# B&R Automation Studio project DeltaTracking
Automation Studio 6.5.1.6; technology packages: mappCockpit 6.3.1, mappMotion 6.6.0, mappView 6.3.0, OpcUaCs 6.0.0

## Configuration Config1

CPU 5APC3100.KBU3-000, AutomationRuntime 6.6.3, Build 11.3.0, Safety 0.0

### Task classes (Cpu.sw)
```
Cyclic#1 (cycle 2000 us, tolerance 0 us):
  APP_Convey <- Conveyor.APP_Conveyor1.prg
  APP_Robot1 <- Robots.APP_Robot1.prg
DataObjects: Arnc0sys, Acp10sys
NcDataObjects: gmcipuc, gmciplog, gmcipfub, gmcipfun, gmciplsm, gmciplbr, gmcipmxd, gmcipvar, gmcipsys, gmcipiec, gmcipesm, gmcipusm, gmcipcsm, gmcipui, gmcipubr, gmcipcbr, gmcipcfg, gmcipus, gmcipmx, Cam
Binaries: McAcpSys, mcdrivelog, udbdef, TCData, mvLoader, arsvcreg, arflatprv, mCoWebSc, McAcpDrv, McAcpSim, McProfGen, McMechSys, arcoal, ashwac, arconfig, asfw, ashwd, iomap, User, Role, sysconf, TraceConfi, Settings, Config_1, Hierarchy, Config, AxisAx_1, Config_2, ComRobot, Config_4, Config_5, Config_3, Config_6, ToolX20, AxesAxX21, GRobot1, GFRobot1, ARobot1, ComRobot1, WorkRobot1, GRobot2, MRobot1, GFRobot2, FeatX21, TrkDevX21, TrkDevConv, AxisAxX25, MecX20, AxesAxX20, WorkX20, FeatX20, DeltaX20, ComFeatX20, DeltaX21, TrkDevX20, vccddbox, vcfile, vccbtn, vcpdvnc, arialbd, vcmgr, vctcal, vcgclass, vcctext, vccnum, vcfntttf, vcdsloc, vccstr, arial, Visu03, vccshape, vcalarm, Visu01, vccdt, vccscale, vcchtml, vcchspot, vccbmp, vccpopup, vcshared, vcxml, vccurl, vcrt, vccslider, Visu02, vcnet, vcclbox, vcbclass, vcdsint, vcpdsw, vccovl, vccline, TCLang, visvc, vccdbox, vcpfar00, vcpfmtcx, vcpfapc, GrpMaster, Users, UsersLogin, TC, Files, DiagWebXs, AlmMaster, AlmHisMain, AlmMain, GrpVMaster, AlmVMaster, CfgPureVir, AxisPS, AxisAxXX1, AxisAxXX2, AxisMaster, MDevXX1, AxVMaster, GrpDevXX1, AlmDevXX1, GrPDevXX4, AlmDevXX4, GrPDevX10, AlmDevX10, AlmDevX20, GrpDevX20, AlmDevX21, GrpDevX21, AlmMBelts, GrpMBelts, AlmDevXX6, GrpDevXX6, AxesVAxX20, vcpfx20, AxisMBelts, MasMBelts, MBeltsPt, AxesVAxX25, AxesAxX10, AxesAxX25, WorkX10, CncXX6, MecX10, AxesVAxX10, DeltaX10, FeatXX6, FeatX10, ToolX10, ToolXX6, MecXX6, MotMaster, MotVMaster, vcctrend, MotDevX10, GrPDevXX3, AlmDevXX3, MotDevXX3, GrPDevXX2, MotDevXX1, AlmDevXX2, MotDevXX2, vcpkat, arnc0cfg, Sdc10map, Arnc0map, Sdc10map1, Sdc10map2, MotDevX20, MotDevX11, MotDevXX9, GrpDevXX9, AlmDevXX9, PML, MotDevXX6, CncDevXX6, MotDevXX7, AlmDevXX7, GrpDevXX7, Robot, AlmDevXX8, GrpDevXX8, MotSim, MotSpindle, MotDevXXA, AlmDevXXA, GrpDevXXA, GrpDevX11, AlmDevX11, OpcUaBasic, User_1, OpcUaMap, AlmHmi, AlmHistHmi, Groups, vccpiech, MotMac, acp10cfg, Acp10map
Libraries: standard, AsBrStr, sys_lib, runtime, AsArSdm, astime, brsystem, FileIO, AsIODiag, DataObj, AsArProf, AsMem, AsIOAcc, AsEPL, ASMcDcs, AsBrMath, visapi, ArTextSys, AsSem, AsIecCon, AsZip, powerlnk, aruser, asusb, ashw, arcert, arssl, aseth, asio, vcresman, IecCheck, areventlog, MpCom, MpUserX, MpFile, MpRecipe, MpAlarmX, MpBase, CoTrace, MpServer, McBase, McAxGroup, McAcpAx, McAxis, McPathGen, McTrkPath, MpAxis, McProgInt, McPureVAx, McDS402Ax, MpRobotics, MpCnc, MpTool
```

### Hardware
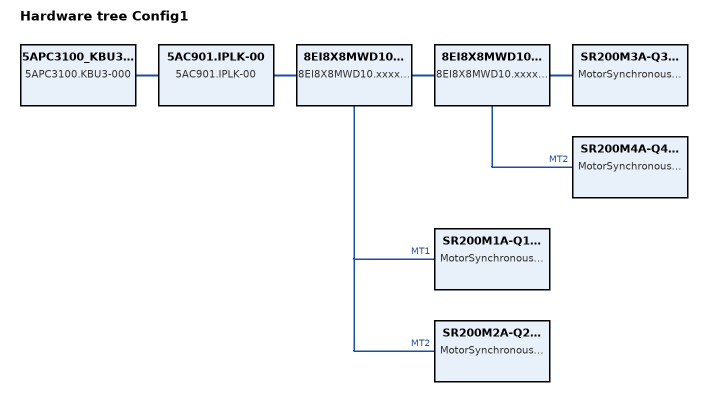
```
5AC901.IPLK-00 : 5AC901.IPLK-00 v2.1.0.0  [SL -> 5APC3100_KBU3_000.SL2]
  Connector IF1:
    DNAConfiguration = manual
    Channel1
    ChannelID1 = McAcpBroadcast
    ChannelType1 = OCTET[96]
5APC3100_KBU3_000 : 5APC3100.KBU3-000 v2.3.1.0
  Connector IF3:
    AssignedOperatingSystem = ARemb
    ActivateDevice = 1
    HostName = apc3100robert
    Mode = Manual
    InternetAddress = 10.43.51.43
    SubnetMask = 255.255.255.0
    Vnc1
    VncKeyMappingFile1 = 
    VncRefreshRate1 = 100
    ActivateSnmp = 2
  Connector IF4:
    AssignedOperatingSystem = ARemb
    ActivateDevice = 1
    HostName = apc3100robert
    Mode = DHCPServer
    InternetAddress = 192.168.20.254
    SubnetMask = 255.255.255.0
    Lease1
    LeaseName1 = Range1
    LeaseStartAddress1 = 192.168.20.100
    LeaseStopAddress1 = 192.168.20.110
    LeaseSubnetMask1 = 255.255.255.0
    Vnc1
    VncTitle1 = VNC
    ActivateSnmp = 2
  Connector IF5:
    AssignedOperatingSystem = ARemb
  Connector IF6:
    AssignedOperatingSystem = ARemb
  Connector IF7:
    AssignedOperatingSystem = ARemb
  Connector IF8:
    AssignedOperatingSystem = ARemb
  ConfigurationID = Template_X20CP1586
  UserPartitionSize = 5
  Simulation = 1
  TimerDeviceType = EPLX2X
  TimerDevice = 5AC901.IPLK-00.IF1
  IdleTaskClass = 4
  TaskClassIdleTime = 4000
  Cyclic1Duration = 2000
  Cyclic1Tolerance = 0
  Cyclic1Stack = 16384
  Cyclic2Duration = 4000
  Cyclic2Tolerance = 0
  Cyclic3Duration = 10000
  Cyclic3Tolerance = 0
  Cyclic4Duration = 20000
  Cyclic4Tolerance = 0
  Cyclic5Duration = 50000
  Cyclic5Tolerance = 0
  Cyclic6Duration = 100000
  Cyclic6Tolerance = 0
  Cyclic7Duration = 200000
  Cyclic7Tolerance = 0
  FileDevice1
  FileDeviceName1 = SceneViewer
  FileDevicePath1 = USER_PATH
  FileDevice2
  FileDeviceName2 = MPLogDir
  FileDevicePath2 = USER_PATH\Log
  FileDevice3
  FileDeviceName3 = DebugData
  FileDevicePath3 = USER_PATH\\Debug
  FileDevice4
  FileDeviceName4 = CNC_PrgDir
  FileDevicePath4 = USER_PATH\CNC_Prg
  EthernetDefaultGateway = 10.43.51.1
  ActivateFtpServer = 1
  FTPProtocol = 2
  FtpUser1
  FtpUsername1 = gmctest
  FtpUserPassword1 = dJg12F/7hd2fGO/QauVo5qNTeUud8LRwkPqca2btE1Q=
  FtpUserSalt1 = iGhlfz5v
  FTPAccessRight1 = 0
  FTPdevice1 = ALL
  ActivateWebServer = 1
  ActivateSdm = 1
8EI8X8MWD10.xxxx-1-Q1-Q2_SRr500_1 : 8EI8X8MWD10.xxxx-1 v2.4.0.0 (NodeNumber=1)  [PLK1 -> 5AC901.IPLK-00.IF1 [Cable Type=PowerlinkCable, Length=10, Version=1.0.0.3]; PLK2 -> 8EI8X8MWD10.xxxx-1-Q3-Q4_SRr500_1.PLK1 [Cable Type=PowerlinkCable, Length=10, Version=1.0.0.3]; MT2 -> SR200M2A-Q2_SRr500_1.MT]
  DriveConfiguration/Encoder/EncoderX41:
    InterfaceType = T_Format
  DriveConfiguration/Encoder/EncoderX42:
    InterfaceType = T_Format
  DriveConfiguration/Channel[1]/RealAxis:
    AxisReference = gAxisQ1_SRr500_1
  DriveConfiguration/Channel[1]/RealAxis/MechanicalElements/Gearbox:
    InputIsReadOnly = 1
    Input = 80
    OutputIsReadOnly = 1
  DriveConfiguration/Channel[1]/RealAxis/MechanicalElements/RotaryToLinearTransformation:
    ReferenceDistanceIsReadOnly = 1
    ReferenceDistance = 360
  DriveConfiguration/Channel[1]/RealAxis/Controller:
    ModeIsReadOnly = 1
    Mode = PositionControllerWithTorqueFeedForward
  DriveConfiguration/Channel[1]/RealAxis/Controller/Mode/Position:
    ProportionalGainIsReadOnly = 1
    ProportionalGain = 60.0
    IntegrationTimeIsReadOnly = 1
  DriveConfiguration/Channel[1]/RealAxis/Controller/Mode/Speed:
    ProportionalGainIsReadOnly = 1
    ProportionalGain = 0.5
    IntegrationTimeIsReadOnly = 1
    FilterTimeIsReadOnly = 1
  DriveConfiguration/Channel[1]/RealAxis/Controller/Mode:
    FeedForwardIsReadOnly = 1
    FeedForward = CyclicValueFromAxesGroup
  DriveConfiguration/Channel[1]/RealAxis/Controller/Mode/LoopFilters:
    LoopFilterXIsReadOnly = 1
  DriveConfiguration/Channel[1]/RealAxis/Homing:
    Mode = AbsoluteCorrection
    RestorePositionVariable = 
  DriveConfiguration/Channel[1]/RealAxis/StopReaction:
    DriveError = CyclicDecelerationFromAxesGroup
  DriveConfiguration/Channel[1]/RealAxis/MovementErrorLimits:
    PositionError = 3.0
  DriveConfiguration/Channel[1]/RealAxis:
    JerkFilterIsReadOnly = 1
    JerkFilter = Used
  DriveConfiguration/Channel[1]/RealAxis/JerkFilter:
    JerkTimeMin = 0.025
    JerkTime = 0.025
  DriveConfiguration/Channel[2]/RealAxis:
    AxisReference = gAxisQ2_SRr500_1
  DriveConfiguration/Channel[2]/RealAxis/MechanicalElements/Gearbox:
    InputIsReadOnly = 1
    Input = 50
    OutputIsReadOnly = 1
  DriveConfiguration/Channel[2]/RealAxis/MechanicalElements/RotaryToLinearTransformation:
    ReferenceDistanceIsReadOnly = 1
    ReferenceDistance = 360
  DriveConfiguration/Channel[2]/RealAxis/Controller:
    ModeIsReadOnly = 1
    Mode = PositionControllerWithTorqueFeedForward
  DriveConfiguration/Channel[2]/RealAxis/Controller/Mode/Position:
    ProportionalGainIsReadOnly = 1
    ProportionalGain = 75.0
    IntegrationTimeIsReadOnly = 1
  DriveConfiguration/Channel[2]/RealAxis/Controller/Mode/Speed:
    ProportionalGainIsReadOnly = 1
    ProportionalGain = 0.5
    IntegrationTimeIsReadOnly = 1
    FilterTimeIsReadOnly = 1
  DriveConfiguration/Channel[2]/RealAxis/Controller/Mode:
    FeedForwardIsReadOnly = 1
    FeedForward = CyclicValueFromAxesGroup
  DriveConfiguration/Channel[2]/RealAxis/Controller/Mode/LoopFilters:
    LoopFilterXIsReadOnly = 1
  DriveConfiguration/Channel[2]/RealAxis/Homing:
    Mode = AbsoluteCorrection
    RestorePositionVariable = 
  DriveConfiguration/Channel[2]/RealAxis/StopReaction:
    DriveError = CyclicDecelerationFromAxesGroup
  DriveConfiguration/Channel[2]/RealAxis/MovementErrorLimits:
    PositionError = 1.0
  DriveConfiguration/Channel[2]/RealAxis:
    JerkFilterIsReadOnly = 1
    JerkFilter = Used
  DriveConfiguration/Channel[2]/RealAxis/JerkFilter:
    JerkTimeMin = 0.025
    JerkTime = 0.025
8EI8X8MWD10.xxxx-1-Q3-Q4_SRr500_1 : 8EI8X8MWD10.xxxx-1 v2.4.0.0 (NodeNumber=2)  [PLK1 -> 8EI8X8MWD10.xxxx-1-Q1-Q2_SRr500_1.PLK2 [Cable Type=PowerlinkCable, Length=10, Version=1.0.0.3]; MT2 -> SR200M4A-Q4_SRr500_1.MT]
  DriveConfiguration/Encoder/EncoderX41:
    InterfaceType = T_Format
  DriveConfiguration/Encoder/EncoderX42:
    InterfaceType = T_Format
  DriveConfiguration/Channel[1]/RealAxis:
    AxisReference = gAxisQ3_SRr500_1
  DriveConfiguration/Channel[1]/RealAxis/MechanicalElements/Gearbox:
    InputIsReadOnly = 1
    Input = 2
    OutputIsReadOnly = 1
    Output = 25
  DriveConfiguration/Channel[1]/RealAxis/MechanicalElements/RotaryToLinearTransformation:
    ReferenceDistanceIsReadOnly = 1
    ReferenceDistance = 1.0
  DriveConfiguration/Channel[1]/RealAxis/Controller:
    ModeIsReadOnly = 1
    Mode = PositionControllerWithTorqueFeedForward
  DriveConfiguration/Channel[1]/RealAxis/Controller/Mode/Position:
    ProportionalGainIsReadOnly = 1
    ProportionalGain = 225.0
    IntegrationTimeIsReadOnly = 1
  DriveConfiguration/Channel[1]/RealAxis/Controller/Mode/Speed:
    ProportionalGainIsReadOnly = 1
    ProportionalGain = 0.6
    IntegrationTimeIsReadOnly = 1
    FilterTimeIsReadOnly = 1
  DriveConfiguration/Channel[1]/RealAxis/Controller/Mode:
    FeedForwardIsReadOnly = 1
    FeedForward = CyclicValueFromAxesGroup
  DriveConfiguration/Channel[1]/RealAxis/Controller/Mode/LoopFilters:
    LoopFilterXIsReadOnly = 1
  DriveConfiguration/Channel[1]/RealAxis/Homing:
    Mode = RestorePosition
    RestorePositionVariable = 
  DriveConfiguration/Channel[1]/RealAxis/StopReaction:
    DriveError = CyclicDecelerationFromAxesGroup
  DriveConfiguration/Channel[1]/RealAxis/MovementErrorLimits:
    PositionError = 1.0
  DriveConfiguration/Channel[1]/RealAxis:
    JerkFilterIsReadOnly = 1
    JerkFilter = Used
  DriveConfiguration/Channel[1]/RealAxis/JerkFilter:
    JerkTimeMin = 0.025
    JerkTime = 0.025
  DriveConfiguration/Channel[1]/RealAxis/AxisFeatures:
    FeatureRef[1] = Feature_Brake_SRr500_1
  DriveConfiguration/Channel[2]/RealAxis:
    AxisReference = gAxisQ4_SRr500_1
  DriveConfiguration/Channel[2]/RealAxis/MechanicalElements/Gearbox:
    InputIsReadOnly = 1
    Input = 1875
    OutputIsReadOnly = 1
    Output = 132
  DriveConfiguration/Channel[2]/RealAxis/MechanicalElements/RotaryToLinearTransformation:
    ReferenceDistanceIsReadOnly = 1
    ReferenceDistance = 360
  DriveConfiguration/Channel[2]/RealAxis/Controller:
    ModeIsReadOnly = 1
    Mode = PositionControllerWithTorqueFeedForward
  DriveConfiguration/Channel[2]/RealAxis/Controller/Mode/Position:
    ProportionalGainIsReadOnly = 1
    ProportionalGain = 200.0
    IntegrationTimeIsReadOnly = 1
  DriveConfiguration/Channel[2]/RealAxis/Controller/Mode/Speed:
    ProportionalGainIsReadOnly = 1
    ProportionalGain = 0.4
    IntegrationTimeIsReadOnly = 1
    FilterTimeIsReadOnly = 1
  DriveConfiguration/Channel[2]/RealAxis/Controller/Mode:
    FeedForwardIsReadOnly = 1
    FeedForward = CyclicValueFromAxesGroup
  DriveConfiguration/Channel[2]/RealAxis/Controller/Mode/LoopFilters:
    LoopFilterXIsReadOnly = 1
  DriveConfiguration/Channel[2]/RealAxis/Homing:
    Mode = RestorePosition
    RestorePositionVariable = 
  DriveConfiguration/Channel[2]/RealAxis/StopReaction:
    DriveError = CyclicDecelerationFromAxesGroup
  DriveConfiguration/Channel[2]/RealAxis/MovementErrorLimits:
    PositionError = 1.0
  DriveConfiguration/Channel[2]/RealAxis:
    JerkFilterIsReadOnly = 1
    JerkFilter = Used
  DriveConfiguration/Channel[2]/RealAxis/JerkFilter:
    JerkTimeMin = 0.025
    JerkTime = 0.025
  DriveConfiguration/Channel[2]/RealAxis/AxisFeatures:
    FeatureRef[1] = Feature_Brake_SRr500_1
SR200M1A-Q1_SRr500_1 : MotorSynchronous_any v2.2.1.0  [MT -> 8EI8X8MWD10.xxxx-1-Q1-Q2_SRr500_1.MT1]
  M1/MotorParameters:
    MOTOR_POLEPAIRS = 5
    MOTOR_SPEED_RATED = 3000
    MOTOR_SPEED_MAX = 6000
    MOTOR_VOLTAGE_RATED = 220
    MOTOR_CURR_RATED = 4.9
    MOTOR_CURR_STALL = 4.9
    MOTOR_CURR_MAX = 17.2
    MOTOR_TORQ_RATED = 1.91
    MOTOR_TORQ_STALL = 1.91
    MOTOR_TORQ_MAX = 6.69
    MOTOR_VOLTAGE_CONST = 26.4
    MOTOR_TORQ_CONST = 0.39
    MOTOR_STATOR_RESISTANCE = 1.3
    MOTOR_STATOR_INDUCTANCE = 2.4
    MOTOR_INERTIA = 0.818
  M1/MotorParameters/EncoderMounting/Angle:
    MOTOR_COMMUT_OFFSET = 3.14
  M1/MotorParameters:
    TemperatureSensor = NotUsed
    TemperatureModel = Current
  M1/MotorParameters/TemperatureModel:
    MOTOR_WIND_TEMP_MAX = 100
    MOTOR_WIND_CROSS_SECT = 0
    MOTOR_TAU_THERM = 100
  M1:
    Encoder = NotUsed
    Gearbox = UsedWithDynamicTorqueLimitation
  M1/Gearbox/GearRatio:
    Input = 80
  M1/Gearbox:
    MOTORGEAR_SPEED_MAX = 5500
    MOTORGEAR_TORQ_NOM = 178
    MOTORGEAR_TORQ_MAX = 178
    MOTORGEAR_INERTIA = 0.532
    MOTORGEAR_VISC_FRIC = 0.0019144080232812802
    MOTORGEAR_STAT_FRIC = 0.16999999999999998
SR200M2A-Q2_SRr500_1 : MotorSynchronous_any v2.2.1.0  [MT -> 8EI8X8MWD10.xxxx-1-Q1-Q2_SRr500_1.MT2]
  M1/MotorParameters:
    MOTOR_POLEPAIRS = 5
    MOTOR_SPEED_RATED = 3000
    MOTOR_SPEED_MAX = 6000
    MOTOR_VOLTAGE_RATED = 220
    MOTOR_CURR_RATED = 2.9
    MOTOR_CURR_STALL = 2.9
    MOTOR_CURR_MAX = 10.2
    MOTOR_TORQ_RATED = 1.27
    MOTOR_TORQ_STALL = 1.27
    MOTOR_TORQ_MAX = 4.46
    MOTOR_VOLTAGE_CONST = 29.3
    MOTOR_TORQ_CONST = 0.439
    MOTOR_STATOR_RESISTANCE = 3.3
    MOTOR_STATOR_INDUCTANCE = 5.2
    MOTOR_INERTIA = 0.45
  M1/MotorParameters/EncoderMounting/Angle:
    MOTOR_COMMUT_OFFSET = 3.14
  M1/MotorParameters:
    TemperatureSensor = NotUsed
    TemperatureModel = Current
  M1/MotorParameters/TemperatureModel:
    MOTOR_WIND_TEMP_MAX = 100
    MOTOR_WIND_CROSS_SECT = 0
    MOTOR_TAU_THERM = 100
  M1:
    Encoder = NotUsed
    Gearbox = UsedWithDynamicTorqueLimitation
  M1/Gearbox/GearRatio:
    Input = 50
  M1/Gearbox:
    MOTORGEAR_SPEED_MAX = 6000
    MOTORGEAR_TORQ_NOM = 73
    MOTORGEAR_TORQ_MAX = 73
    MOTORGEAR_INERTIA = 0.20
    MOTORGEAR_VISC_FRIC = 0.001198831756609865
    MOTORGEAR_STAT_FRIC = 0.1
SR200M3A-Q3_SRr500_1 : MotorSynchronous_any v2.2.1.0  [MT -> 8EI8X8MWD10.xxxx-1-Q3-Q4_SRr500_1.MT1]
  M1/MotorParameters:
    MOTOR_POLEPAIRS = 5
    MOTOR_SPEED_RATED = 3000
    MOTOR_SPEED_MAX = 6000
    MOTOR_VOLTAGE_RATED = 220
    MOTOR_CURR_RATED = 1.45
    MOTOR_CURR_STALL = 1.45
    MOTOR_CURR_MAX = 5.08
    MOTOR_TORQ_RATED = 0.48
    MOTOR_TORQ_STALL = 0.48
    MOTOR_TORQ_MAX = 1.67
    MOTOR_VOLTAGE_CONST = 23.7
    MOTOR_TORQ_CONST = 0.329
    MOTOR_STATOR_RESISTANCE = 13.6
    MOTOR_STATOR_INDUCTANCE = 9.7
    MOTOR_INERTIA = 0.098
  M1/MotorParameters/EncoderMounting/Angle:
    MOTOR_COMMUT_OFFSET = 3.14
  M1/MotorParameters:
    TemperatureSensor = NotUsed
    TemperatureModel = Current
  M1/MotorParameters/TemperatureModel:
    MOTOR_WIND_TEMP_MAX = 100
    MOTOR_WIND_CROSS_SECT = 0
    MOTOR_TAU_THERM = 100
  M1:
    Brake = Used
  M1/Brake:
    MOTOR_BRAKE_CURR_RATED = 0
    MOTOR_BRAKE_TORQ_RATED = 0.32
    MOTOR_BRAKE_ON_TIME = 0.02
    MOTOR_BRAKE_OFF_TIME = 0.2
    MOTOR_BRAKE_INERTIA = 0.156
  M1:
    Encoder = NotUsed
SR200M4A-Q4_SRr500_1 : MotorSynchronous_any v2.2.1.0  [MT -> 8EI8X8MWD10.xxxx-1-Q3-Q4_SRr500_1.MT2]
  M1/MotorParameters:
    MOTOR_POLEPAIRS = 5
    MOTOR_SPEED_RATED = 3000
    MOTOR_SPEED_MAX = 6000
    MOTOR_VOLTAGE_RATED = 220
    MOTOR_CURR_RATED = 1
    MOTOR_CURR_STALL = 1
    MOTOR_CURR_MAX = 3.4
    MOTOR_TORQ_RATED = 0.3
    MOTOR_TORQ_STALL = 0.3
    MOTOR_TORQ_MAX = 1.1
    MOTOR_VOLTAGE_CONST = 21.3
    MOTOR_TORQ_CONST = 0.3
    MOTOR_STATOR_RESISTANCE = 23.5
    MOTOR_STATOR_INDUCTANCE = 18.1
    MOTOR_INERTIA = 0.1
  M1/MotorParameters/EncoderMounting/Angle:
    MOTOR_COMMUT_OFFSET = 3.14
  M1/MotorParameters:
    TemperatureSensor = NotUsed
    TemperatureModel = Current
  M1/MotorParameters/TemperatureModel:
    MOTOR_WIND_TEMP_MAX = 100
    MOTOR_WIND_CROSS_SECT = 0
    MOTOR_TAU_THERM = 100
  M1:
    Brake = Used
  M1/Brake:
    MOTOR_BRAKE_CURR_RATED = 0
    MOTOR_BRAKE_TORQ_RATED = 0.32
    MOTOR_BRAKE_ON_TIME = 0.02
    MOTOR_BRAKE_OFF_TIME = 0.2
    MOTOR_BRAKE_INERTIA = 0.156
  M1:
    Encoder = NotUsed
```

### Config_10.mechanicalsystem - 5APC3100_KBU3_000/mappMotion/Codian_SRr500_1/Config_10.mechanicalsystem
```
Element MechSys_SRr500_1 (Type=mechanicalsystem)  // Codian SR200-6/500Z20A [RobotID="CodianSR200p6r500Z20A" Version="6.8.0"]
  TypeIsReadOnly = 1
  Type = Scara
    SubtypeIsReadOnly = 1
    Subtype:
      SceneViewerObject = ObjectID
        ID = 2710
      DescriptionIsReadOnly = 1
      Description:
        Dimensions:
          TranslationFromBaseToQ1IsReadOnly = 1
          TranslationFromBaseToQ1:
            Z = 177.0
          TranslationFromQ1ToQ2IsReadOnly = 1
          TranslationFromQ1ToQ2:
            XY = 225.0
            Z = 54.5
          TranslationFromQ2ToQZ:
            XY = 275.0
          TranslationFromQZToQCIsReadOnly = 1
          TranslationFromQZToQC:
            Z = -53.5
          TranslationFromQCToFlangeIsReadOnly = 1
          TranslationFromQCToFlange:
            Z = -30.0
        Offsets:
          JointAxisIsReadOnly = 1
          JointAxis[1]
          JointAxis[2]
          JointAxis[3]
          JointAxis[4]
        CountDirections:
          JointAxisIsReadOnly = 1
          JointAxis[1]
          JointAxis[2]
          JointAxis[3]
          JointAxis[4]
      TcpOrientation:
        Frames = Used
      WireFrameModel:
        Q1ToQ2:
          Distance = 5.0
        Q2ToQZ:
          Distance = 5.0
        QZToQC:
          Distance = 5.0
        QCToFlange:
          Distance = 5.0
        FlangeToTcp:
          Distance = 5.0
      DynamicModelIsReadOnly = 1
      InternalDynamicModelIsReadOnly = 1
      InternalDynamicModel = Used
        TypeIsReadOnly = 1
        Type = Codian SR200-6/500Z20A
        Row[1]:
          Value = 6
          Unit = 
          Description = Dynamic_model_variant
        Row[2]:
          Index = 1
          Value = 3.791755
          Unit = kg
          Description = m1
        Row[3]:
          Index = 2
          Value = 0.573779741865
          Unit = kgm
          Description = m1*rc1x
        Row[4]:
          Index = 3
          Value = 0.00049292815
          Unit = kgm
          Description = m1*rc1y
        Row[5]:
          Index = 4
          Value = 0.20037908473
          Unit = kgm
          Description = m1*rc1z
        Row[6]:
          Index = 5
          Value = 0.0000745913664424
          Unit = kgm²
          Description = m1*rc1x*rc1y
        Row[7]:
          Index = 6
          Value = 0.0000260492810149
          Unit = kgm²
          Description = m1*rc1y*rc1z
        Row[8]:
          Index = 7
          Value = 0.0303219642386
          Unit = kgm²
          Description = m1*rc1x*rc1z
        Row[9]:
          Index = 8
          Value = 0.0868260718782
          Unit = kgm²
          Description = m1*rc1x*rc1x
        Row[10]:
          Index = 9
          Value = 0.0000000640806595
          Unit = kgm²
          Description = m1*rc1y*rc1y
        Row[11]:
          Index = 10
          Value = 0.0105892331116
          Unit = kgm²
          Description = m1*rc1z*rc1z
        Row[12]:
          Index = 11
          Value = 0.019199
          Unit = kgm²
          Description = Jxx1
        Row[13]:
          Index = 12
          Value = 0.136703
          Unit = kgm²
          Description = Jyy1
        Row[14]:
          Index = 13
          Value = 0.123126
          Unit = kgm²
          Description = Jzz1
        Row[15]:
          Index = 14
          Value = 4.530055
          Unit = kg
          Description = m2
        Row[16]:
          Index = 15
          Value = 0.3856888827
          Unit = kgm
          Description = m2*rc2x
        Row[17]:
          Index = 16
          Value = 0.00221972695
          Unit = kgm
          Description = m2*rc2y
        Row[18]:
          Index = 17
          Value = 0.320632762845
          Unit = kgm
          Description = m2*rc2z
        Row[19]:
          Index = 18
          Value = 0.000188987552523
          Unit = kgm²
          Description = m2*rc2x*rc2y
        Row[20]:
          Index = 19
          Value = 0.000157110053794
          Unit = kgm²
          Description = m2*rc2y*rc2z
        Row[21]:
          Index = 20
          Value = 0.0272986734286
          Unit = kgm²
          Description = m2*rc2x*rc2z
        Row[22]:
          Index = 21
          Value = 0.0328375514731
          Unit = kgm²
          Description = m2*rc2x*rc2x
        Row[23]:
          Index = 22
          Value = 0.0000010876662055
          Unit = kgm²
          Description = m2*rc2y*rc2y
        Row[24]:
          Index = 23
          Value = 0.0226940663214
          Unit = kgm²
          Description = m2*rc2z*rc2z
        Row[25]:
          Index = 24
          Value = 0.053513
          Unit = kgm²
          Description = Jxx2
        Row[26]:
          Index = 25
          Value = 0.167955
          Unit = kgm²
          Description = Jyy2
        Row[27]:
          Index = 26
          Value = 0.126363
          Unit = kgm²
          Description = Jzz2
        Row[28]:
          Index = 27
          Unit = kg
          Description = m3
        Row[29]:
          Index = 28
          Unit = kgm
          Description = m3*rc3x
        Row[30]:
          Index = 29
          Unit = kgm
          Description = m3*rc3y
        Row[31]:
          Index = 30
          Unit = kgm
          Description = m3*rc3z
        Row[32]:
          Index = 31
          Unit = kgm²
          Description = m3*rc3x*rc3y
        Row[33]:
          Index = 32
          Unit = kgm²
          Description = m3*rc3y*rc3z
        Row[34]:
          Index = 33
          Unit = kgm²
          Description = m3*rc3x*rc3z
        Row[35]:
          Index = 34
          Unit = kgm²
          Description = m3*rc3x*rc3x
        Row[36]:
          Index = 35
          Unit = kgm²
          Description = m3*rc3y*rc3y
        Row[37]:
          Index = 36
          Unit = kgm²
          Description = m3*rc3z*rc3z
        Row[38]:
          Index = 37
          Unit = kgm²
          Description = Jxx3
        Row[39]:
          Index = 38
          Unit = kgm²
          Description = Jyy3
        Row[40]:
          Index = 39
          Unit = kgm²
          Description = Jzz3
        Row[41]:
          Index = 40
          Value = 0.859593
          Unit = kg
          Description = m4
        Row[42]:
          Index = 41
          Unit = kgm
          Description = m4*rc4x
        Row[43]:
          Index = 42
          Unit = kgm
          Description = m4*rc4y
        Row[44]:
          Index = 43
          Value = 0.058762637073
          Unit = kgm
          Description = m4*rc4z
        Row[45]:
          Index = 44
          Unit = kgm²
          Description = m4*rc4x*rc4y
        Row[46]:
          Index = 45
          Unit = kgm²
          Description = m4*rc4y*rc4z
        Row[47]:
          Index = 46
          Unit = kgm²
          Description = m4*rc4x*rc4z
        Row[48]:
          Index = 47
          Unit = kgm²
          Description = m4*rc4x*rc4x
        Row[49]:
          Index = 48
          Unit = kgm²
          Description = m4*rc4y*rc4y
        Row[50]:
          Index = 49
          Value = 0.00401707263295
          Unit = kgm²
          Description = m4*rc4z*rc4z
        Row[51]:
          Index = 50
          Unit = kgm²
          Description = Jxx4
        Row[52]:
          Index = 51
          Unit = kgm²
          Description = Jyy4
        Row[53]:
          Index = 52
          Value = 0.000371
          Unit = kgm²
          Description = Jzz4
        Row[54]:
          Index = 53
          Value = 0.000135
          Unit = kgm²
          Description = JMotor1
        Row[55]:
          Index = 54
          Value = 0.000065
          Unit = kgm²
          Description = JMotor2
        Row[56]:
          Index = 55
          Value = 0.000055
          Unit = kgm²
          Description = JMotor3
        Row[57]:
          Index = 56
          Value = 0.00003
          Unit = kgm²
          Description = JMotor4
        Row[58]:
          Index = 57
          Value = 1.95
          Unit = Nms
          Description = dV1
        Row[59]:
          Index = 58
          Value = 0.477
          Unit = Nms
          Description = dV2
        Row[60]:
          Index = 59
          Value = 120.0
          Unit = Ns/m
          Description = dV3
        Row[61]:
          Index = 60
          Value = 0.0129
          Unit = Nms
          Description = dV4
        Row[62]:
          Index = 61
          Value = 13.6
          Unit = Nm
          Description = dC1
        Row[63]:
          Index = 62
          Value = 5.0
          Unit = Nm
          Description = dC2
        Row[64]:
          Index = 63
          Value = 35.0
          Unit = N
          Description = dC3
        Row[65]:
          Index = 64
          Value = 0.37
          Unit = Nm
          Description = dC4
      InternalDynamicLimits = Used
        TypeIsReadOnly = 1
        Type = Codian SR200-6/500Z20A
        GearboxLimits:
          Row[1]:
            Value = 6
            Unit = Variant
            Description = Variant of dynamic model
          Row[2]:
            Index = 1
            Value = 113.0
            Unit = Nm
            Description = Gearbox Drive 1 Output Torque Limit
          Row[3]:
            Index = 2
            Value = 44.0
            Unit = Nm
            Description = Gearbox Drive 2 Output Torque Limit
          Row[4]:
            Index = 3
            Value = 100.0
            Unit = Nm
            Description = Gearbox Drive 3 Output Torque Limit
          Row[5]:
            Index = 4
            Value = 1.3
            Unit = Nm
            Description = Gearbox Drive 4 Output Torque Limit
      ConditionalLimitReduction4Ax = Used
        ConditionalLimitReductionList4Ax[1] = ConditionReductionU
          LimitReductionInfluence4Ax:
            LimitRedInfluenceList[1] = Yes
            LimitRedInfluenceList[2]
            LimitRedInfluenceList[3]
            LimitRedInfluenceList[4]
          CondLimRedPoint[1]:
            SourceValue = 0.0
            LimitReductionInPercent = 0.0
          CondLimRedPoint[2]:
            SourceValue = 2.0
            LimitReductionInPercent = 0.0
          CondLimRedPoint[3]:
            SourceValue = 4.0
            LimitReductionInPercent = 40.0
          CondLimRedPoint[4]:
            SourceValue = 6.0
            LimitReductionInPercent = 65.0
          CondLimRedPoint[5]
          CondLimRedPoint[6]
          CondLimRedPoint[7]
          CondLimRedPoint[8]
          CondLimRedPoint[9]
          CondLimRedPoint[10]
        ConditionalLimitReductionList4Ax[2] = ConditionReductionU
          LimitReductionInfluence4Ax:
            LimitRedInfluenceList[1]
            LimitRedInfluenceList[2] = Yes
            LimitRedInfluenceList[3]
            LimitRedInfluenceList[4]
          CondLimRedPoint[1]:
            SourceValue = 0.0
            LimitReductionInPercent = 0.0
          CondLimRedPoint[2]:
            SourceValue = 2.0
            LimitReductionInPercent = 0.0
          CondLimRedPoint[3]:
            SourceValue = 4.0
            LimitReductionInPercent = 54.0
          CondLimRedPoint[4]:
            SourceValue = 6.0
            LimitReductionInPercent = 70.0
          CondLimRedPoint[5]
          CondLimRedPoint[6]
          CondLimRedPoint[7]
          CondLimRedPoint[8]
          CondLimRedPoint[9]
          CondLimRedPoint[10]
        ConditionalLimitReductionList4Ax[3] = ConditionReductionU
          LimitReductionInfluence4Ax:
            LimitRedInfluenceList[1]
            LimitRedInfluenceList[2]
            LimitRedInfluenceList[3] = Yes
            LimitRedInfluenceList[4]
          CondLimRedPoint[1]:
            SourceValue = 0.0
            LimitReductionInPercent = 0.0
          CondLimRedPoint[2]:
            SourceValue = 2.0
            LimitReductionInPercent = 0.0
          CondLimRedPoint[3]:
            SourceValue = 4.0
            LimitReductionInPercent = 54.0
          CondLimRedPoint[4]:
            SourceValue = 6.0
            LimitReductionInPercent = 83.0
          CondLimRedPoint[5]
          CondLimRedPoint[6]
          CondLimRedPoint[7]
          CondLimRedPoint[8]
          CondLimRedPoint[9]
          CondLimRedPoint[10]
        ConditionalLimitReductionList4Ax[4]
        ConditionalLimitReductionList4Ax[5]
      Couplings:
        LinearCoupling[1]:
          SourceAxisIsReadOnly = 1
          SourceAxis = 4
          SourceAxisUnitsIsReadOnly = 1
          SourceAxisUnits = 360.0
          TargetJointAxisIsReadOnly = 1
          TargetJointAxis = 3
          TargetJointAxisUnitsIsReadOnly = 1
          TargetJointAxisUnits = 20.0
      JointAxesPositionLimits:
        SingleJointAxisIsReadOnly[1] = 1
        SingleJointAxisIsReadOnly[2] = 1
        SingleJointAxisIsReadOnly[3] = 1
        SingleJointAxisIsReadOnly[4]
        JointAxis[1] = ConfigureJointAxesLimits
          LowerLimitMin = -132.0
          UpperLimitMax = 132.0
          LowerLimit = -132.0
          UpperLimit = 132.0
        JointAxis[2] = ConfigureJointAxesLimits
          LowerLimitMin = -150.0
          UpperLimitMax = 150.0
          LowerLimit = -150.0
          UpperLimit = 150.0
        JointAxis[3] = ConfigureJointAxesLimits
          LowerLimitMin = -190.0
          UpperLimitMax = 10.0
          LowerLimit = -190.0
          UpperLimit = 10.0
        JointAxis[4]
      MonitoringPoints = Standard
```

### Config_12.axesgroupfeature - 5APC3100_KBU3_000/mappMotion/Codian_SRr500_1/Config_12.axesgroupfeature
```
Element Feature_Programs_SRr500_1 (Type=axesgroupfeature)  // Codian SR200-6/500Z20A [RobotID="CodianSR200p6r500Z20A" Version="6.8.0"]
  Type:
    InitialSettings:
      AccuracyHoldDelays = User defined
        UserAxesDelay = 0.025
Element Feature_Jogging_SRr500_1 (Type=axesgroupfeature)  // Codian SR200-6/500Z20A [RobotID="CodianSR200p6r500Z20A" Version="6.8.0"]
  Type = Jogging
Element Feature_FeedForward_SRr500_1 (Type=axesgroupfeature)  // Codian SR200-6/500Z20A [RobotID="CodianSR200p6r500Z20A" Version="6.8.0"]
  Type = FeedForward
    RiseTime = 0.25
    Filter = AxisJerkTime
Element Feature_SharedBrakesSignals_SRr500_1 (Type=axesgroupfeature)  // Codian SR200-6/500Z20A [RobotID="CodianSR200p6r500Z20A" Version="6.8.0"]
  Type = SharedBrakesSignals
    BrakeComposite[1]:
      Axes:
        AxisRef[1] = gAxisQ3_SRr500_1
        AxisRef[2] = gAxisQ4_SRr500_1
      Output:
        AxisRef = gAxisQ4_SRr500_1
      Feedback:
        ActivationDelay = 0.08
        ReleaseDelay = 0.2
```

### Config_13.axisfeature - 5APC3100_KBU3_000/mappMotion/Codian_SRr500_1/Config_13.axisfeature
```
Element Feature_Brake_SRr500_1 (Type=axisfeature)  // Codian SR200-6/500Z20A [RobotID="CodianSR200p6r500Z20A" Version="6.8.0"]
  Type = Brake
    BrakeControlType:
      ControlMode = External
        CommandAcceptance = Any
      ControlMonitoring = NotUsed
      MovementMonitoring = NotUsed
```

### Config_8.axesgroup - 5APC3100_KBU3_000/mappMotion/Codian_SRr500_1/Config_8.axesgroup
```
Element gAxesGroup_SRr500_1 (Type=axesgroup)  // Codian SR200-6/500Z20A [RobotID="CodianSR200p6r500Z20A" Version="6.8.0"]
  Type = PathGenAxesGroup
    ProcessingTaskClass = 1
    PhysicalAxes:
      JointAxes:
        JointAxis[1]:
          AxisRef = gAxisQ1_SRr500_1
        JointAxis[2]:
          AxisRef = gAxisQ2_SRr500_1
        JointAxis[3]:
          Name = QZ
          AxisRef = gAxisQ3_SRr500_1
        JointAxis[4]:
          Name = QC
          AxisRef = gAxisQ4_SRr500_1
    MechanicalSystem:
      MechSysRef = MechSys_SRr500_1
    BasicSettings:
      GeometryPlanning:
        Rounding:
          SymmetricRounding = No
          LastSegment = Whole
          AvoidZeroCurvature = Yes
          NonCartesianRounding = Yes
        MaxTangentialTransitionDeviation = 0.05
      TrajectoryPlanning:
        LimitCheckResolution:
          Time = 0.005
        BufferTime:
          Time = 0.05
        TorqueLimitConsideration = Approximation
      Miscellaneous:
        TimeStretchOverride:
          JerkSuppression = Basic
            AdaptationTime = 0.3
    StopReaction:
      AxisError:
        AxisReaction = DynamicStop
    AxesGroupFeatures:
      FeatureRef[1] = Feature_Programs
      FeatureRef[2] = Feature_Jogging_SRr500_1
      FeatureRef[3] = Feature_FeedForward_SRr500_1
      FeatureRef[4] = Feature_SharedBrakesSignals_SRr500_1
      FeatureRef[5] = Feature_FrameHierachy
      FeatureRef[6] = Feature_MFunctions
      FeatureRef[7] = Feature_Selection
      FeatureRef[8] = Feature_TrackingRobot
      FeatureRef[9] = Feature_Workspace
      FeatureRef[10] = Feature_PathDefRobot
```

### Config_9.axis - 5APC3100_KBU3_000/mappMotion/Codian_SRr500_1/Config_9.axis
```
Element gAxisQ1_SRr500_1 (Type=axis)  // Codian SR200-6/500Z20A [RobotID="CodianSR200p6r500Z20A" Version="6.8.0"]
  BaseTypeIsReadOnly = 1
  BaseType = RotaryBounded
    MeasurementUnitIsReadOnly = 1
    MeasurementResolutionIsReadOnly = 1
    MeasurementResolution = 0.001
    CountDirectionIsReadOnly = 1
    CountDirection = Inverse
  MovementLimitsIsReadOnly = 1
  MovementLimits = InternalForPathControlledAxis
    Position:
      LowerLimitMin = -132.0
      UpperLimitMax = 132.0
      LowerLimit = -132.0
      UpperLimit = 132.0
    VelocityIsReadOnly = 1
    Velocity:
      VelocityMax = 410.0
      Velocity = 410.0
    AccelerationIsReadOnly = 1
    Acceleration:
      AccelerationMax = 30000.0
      Acceleration = 30000.0
    DecelerationIsReadOnly = 1
    Deceleration:
      DecelerationMax = 30000.0
      Deceleration = 30000.0
    JerkIsReadOnly = 1
    Jerk = Advanced
      JerkAccelerationPositiveMin = 0.0
      JerkAccelerationPositiveMax = 1000000.0
      JerkAccelerationPositive = 1000000.0
      JerkAccelerationNegativeMin = 0.0
      JerkAccelerationNegativeMax = 1000000.0
      JerkAccelerationNegative = 1000000.0
      JerkDecelerationPositiveMin = 0.0
      JerkDecelerationPositiveMax = 1000000.0
      JerkDecelerationPositive = 1000000.0
      JerkDecelerationNegativeMin = 0.0
      JerkDecelerationNegativeMax = 1000000.0
      JerkDecelerationNegative = 1000000.0
    TorqueIsReadOnly = 1
    Torque = Basic
      TorqueMax = 6.69
      Torque = 6.69
Element gAxisQ2_SRr500_1 (Type=axis)  // Codian SR200-6/500Z20A [RobotID="CodianSR200p6r500Z20A" Version="6.8.0"]
  BaseTypeIsReadOnly = 1
  BaseType = RotaryBounded
    MeasurementUnitIsReadOnly = 1
    MeasurementResolutionIsReadOnly = 1
    MeasurementResolution = 0.001
    CountDirectionIsReadOnly = 1
    CountDirection = Inverse
  MovementLimitsIsReadOnly = 1
  MovementLimits = InternalForPathControlledAxis
    Position:
      LowerLimitMin = -150.0
      UpperLimitMax = 150.0
      LowerLimit = -150.0
      UpperLimit = 150.0
    VelocityIsReadOnly = 1
    Velocity:
      VelocityMax = 700.0
      Velocity = 700.0
    AccelerationIsReadOnly = 1
    Acceleration:
      AccelerationMax = 30000.0
      Acceleration = 30000.0
    DecelerationIsReadOnly = 1
    Deceleration:
      DecelerationMax = 30000.0
      Deceleration = 30000.0
    JerkIsReadOnly = 1
    Jerk = Advanced
      JerkAccelerationPositiveMin = 0.0
      JerkAccelerationPositiveMax = 1500000.0
      JerkAccelerationPositive = 1500000.0
      JerkAccelerationNegativeMin = 0.0
      JerkAccelerationNegativeMax = 1500000.0
      JerkAccelerationNegative = 1500000.0
      JerkDecelerationPositiveMin = 0.0
      JerkDecelerationPositiveMax = 1500000.0
      JerkDecelerationPositive = 1500000.0
      JerkDecelerationNegativeMin = 0.0
      JerkDecelerationNegativeMax = 1500000.0
      JerkDecelerationNegative = 1500000.0
    TorqueIsReadOnly = 1
    Torque = Basic
      TorqueMax = 4.46
      Torque = 4.46
Element gAxisQ3_SRr500_1 (Type=axis)  // Codian SR200-6/500Z20A [RobotID="CodianSR200p6r500Z20A" Version="6.8.0"]
  BaseTypeIsReadOnly = 1
  BaseType = Linear
    MeasurementResolutionIsReadOnly = 1
    MeasurementResolution = 0.001
    CountDirectionIsReadOnly = 1
  MovementLimitsIsReadOnly = 1
  MovementLimits = InternalForPathControlledAxis
    VelocityIsReadOnly = 1
    Velocity:
      VelocityMax = 1000.0
    AccelerationIsReadOnly = 1
    Acceleration:
      AccelerationMax = 50000.0
      Acceleration = 50000.0
    DecelerationIsReadOnly = 1
    Deceleration:
      DecelerationMax = 50000.0
      Deceleration = 50000.0
    JerkIsReadOnly = 1
    Jerk = Advanced
      JerkAccelerationPositiveMin = 0.0
      JerkAccelerationPositiveMax = 1500000.0
      JerkAccelerationPositive = 1500000.0
      JerkAccelerationNegativeMin = 0.0
      JerkAccelerationNegativeMax = 1500000.0
      JerkAccelerationNegative = 1500000.0
      JerkDecelerationPositiveMin = 0.0
      JerkDecelerationPositiveMax = 1500000.0
      JerkDecelerationPositive = 1500000.0
      JerkDecelerationNegativeMin = 0.0
      JerkDecelerationNegativeMax = 1500000.0
      JerkDecelerationNegative = 1500000.0
    TorqueIsReadOnly = 1
    Torque = Basic
      TorqueMax = 1.67
      Torque = 1.67
Element gAxisQ4_SRr500_1 (Type=axis)  // Codian SR200-6/500Z20A [RobotID="CodianSR200p6r500Z20A" Version="6.8.0"]
  BaseTypeIsReadOnly = 1
  BaseType = Rotary
    MeasurementUnitIsReadOnly = 1
    MeasurementResolutionIsReadOnly = 1
    MeasurementResolution = 0.001
    CountDirectionIsReadOnly = 1
    CountDirection = Inverse
  MovementLimitsIsReadOnly = 1
  MovementLimits = InternalForPathControlledAxis
    VelocityIsReadOnly = 1
    Velocity:
      VelocityMax = 2000.0
      Velocity = 2000.0
    AccelerationIsReadOnly = 1
    Acceleration:
      AccelerationMax = 30000.0
      Acceleration = 30000.0
    DecelerationIsReadOnly = 1
    Deceleration:
      DecelerationMax = 30000.0
      Deceleration = 30000.0
    JerkIsReadOnly = 1
    Jerk = Advanced
      JerkAccelerationPositiveMin = 0.0
      JerkAccelerationPositiveMax = 2000000.0
      JerkAccelerationPositive = 2000000.0
      JerkAccelerationNegativeMin = 0.0
      JerkAccelerationNegativeMax = 2000000.0
      JerkAccelerationNegative = 2000000.0
      JerkDecelerationPositiveMin = 0.0
      JerkDecelerationPositiveMax = 2000000.0
      JerkDecelerationPositive = 2000000.0
      JerkDecelerationNegativeMin = 0.0
      JerkDecelerationNegativeMax = 2000000.0
      JerkDecelerationNegative = 2000000.0
    TorqueIsReadOnly = 1
    Torque = Basic
      TorqueMax = 1.11
      Torque = 1.11
```

### Config_11.axisfeature - 5APC3100_KBU3_000/mappMotion/Codian_SRr700_1/Config_11.axisfeature
```
Element Feature_Brake_SRr700_1 (Type=axisfeature)  // Codian SR200-6/700Z20A [RobotID="CodianSR200p6r700Z20A" Version="6.8.0"]
  Type = Brake
    BrakeControlType:
      ControlMode = External
        CommandAcceptance = Any
      ControlMonitoring = NotUsed
      MovementMonitoring = NotUsed
```

### Config_2.axesgroup - 5APC3100_KBU3_000/mappMotion/Codian_SRr700_1/Config_2.axesgroup
```
Element gAxesGroup_SRr700_1 (Type=axesgroup)  // Codian SR200-6/700Z20A [RobotID="CodianSR200p6r700Z20A" Version="6.8.0"]
  Type = PathGenAxesGroup
    ProcessingTaskClass = 1
    PhysicalAxes:
      JointAxes:
        JointAxis[1]:
          AxisRef = gAxisQ1_SRr700_1
        JointAxis[2]:
          AxisRef = gAxisQ2_SRr700_1
        JointAxis[3]:
          Name = QZ
          AxisRef = gAxisQ3_SRr700_1
        JointAxis[4]:
          Name = QC
          AxisRef = gAxisQ4_SRr700_1
    MechanicalSystem:
      MechSysRef = MechSys_SRr700_1
    BasicSettings:
      GeometryPlanning:
        Rounding:
          SymmetricRounding = No
          LastSegment = Whole
          AvoidZeroCurvature = Yes
          NonCartesianRounding = Yes
        MaxTangentialTransitionDeviation = 0.05
      TrajectoryPlanning:
        LimitCheckResolution:
          Time = 0.005
        BufferTime:
          Time = 0.05
        TorqueLimitConsideration = Approximation
      Miscellaneous:
        TimeStretchOverride:
          JerkSuppression = Basic
            AdaptationTime = 0.3
    StopReaction:
      AxisError:
        AxisReaction = DynamicStop
    AxesGroupFeatures:
      FeatureRef[1] = Feature_Programs
      FeatureRef[2] = Feature_FeedForward_SRr700_1
      FeatureRef[3] = Feature_SharedBrakesSignals_SRr700_1
      FeatureRef[4] = Feature_MFunctions
      FeatureRef[5] = Feature_PathDefRobot
      FeatureRef[6] = Feature_Selection
      FeatureRef[7] = Feature_TrackingRobot
```

### Config_3.axis - 5APC3100_KBU3_000/mappMotion/Codian_SRr700_1/Config_3.axis
```
Element gAxisQ1_SRr700_1 (Type=axis)  // Codian SR200-6/700Z20A [RobotID="CodianSR200p6r700Z20A" Version="6.8.0"]
  BaseTypeIsReadOnly = 1
  BaseType = RotaryBounded
    MeasurementUnitIsReadOnly = 1
    MeasurementResolutionIsReadOnly = 1
    MeasurementResolution = 0.001
    CountDirectionIsReadOnly = 1
    CountDirection = Inverse
  MovementLimitsIsReadOnly = 1
  MovementLimits = InternalForPathControlledAxis
    Position:
      LowerLimitMin = -132.0
      UpperLimitMax = 132.0
      LowerLimit = -132.0
      UpperLimit = 132.0
    VelocityIsReadOnly = 1
    Velocity:
      VelocityMax = 410.0
      Velocity = 410.0
    AccelerationIsReadOnly = 1
    Acceleration:
      AccelerationMax = 30000.0
      Acceleration = 30000.0
    DecelerationIsReadOnly = 1
    Deceleration:
      DecelerationMax = 30000.0
      Deceleration = 30000.0
    JerkIsReadOnly = 1
    Jerk = Advanced
      JerkAccelerationPositiveMin = 0.0
      JerkAccelerationPositiveMax = 1200000.0
      JerkAccelerationPositive = 1200000.0
      JerkAccelerationNegativeMin = 0.0
      JerkAccelerationNegativeMax = 1200000.0
      JerkAccelerationNegative = 1200000.0
      JerkDecelerationPositiveMin = 0.0
      JerkDecelerationPositiveMax = 1200000.0
      JerkDecelerationPositive = 1200000.0
      JerkDecelerationNegativeMin = 0.0
      JerkDecelerationNegativeMax = 1200000.0
      JerkDecelerationNegative = 1200000.0
    TorqueIsReadOnly = 1
    Torque = Basic
      TorqueMax = 6.69
      Torque = 6.69
Element gAxisQ2_SRr700_1 (Type=axis)  // Codian SR200-6/700Z20A [RobotID="CodianSR200p6r700Z20A" Version="6.8.0"]
  BaseTypeIsReadOnly = 1
  BaseType = RotaryBounded
    MeasurementUnitIsReadOnly = 1
    MeasurementResolutionIsReadOnly = 1
    MeasurementResolution = 0.001
    CountDirectionIsReadOnly = 1
    CountDirection = Inverse
  MovementLimitsIsReadOnly = 1
  MovementLimits = InternalForPathControlledAxis
    Position:
      LowerLimitMin = -150.0
      UpperLimitMax = 150.0
      LowerLimit = -150.0
      UpperLimit = 150.0
    VelocityIsReadOnly = 1
    Velocity:
      VelocityMax = 700.0
      Velocity = 700.0
    AccelerationIsReadOnly = 1
    Acceleration:
      AccelerationMax = 30000.0
      Acceleration = 30000.0
    DecelerationIsReadOnly = 1
    Deceleration:
      DecelerationMax = 30000.0
      Deceleration = 30000.0
    JerkIsReadOnly = 1
    Jerk = Advanced
      JerkAccelerationPositiveMin = 0.0
      JerkAccelerationPositiveMax = 1300000.0
      JerkAccelerationPositive = 1300000.0
      JerkAccelerationNegativeMin = 0.0
      JerkAccelerationNegativeMax = 1300000.0
      JerkAccelerationNegative = 1300000.0
      JerkDecelerationPositiveMin = 0.0
      JerkDecelerationPositiveMax = 1300000.0
      JerkDecelerationPositive = 1300000.0
      JerkDecelerationNegativeMin = 0.0
      JerkDecelerationNegativeMax = 1300000.0
      JerkDecelerationNegative = 1300000.0
    TorqueIsReadOnly = 1
    Torque = Basic
      TorqueMax = 4.46
      Torque = 4.46
Element gAxisQ3_SRr700_1 (Type=axis)  // Codian SR200-6/700Z20A [RobotID="CodianSR200p6r700Z20A" Version="6.8.0"]
  BaseTypeIsReadOnly = 1
  BaseType = Linear
    MeasurementResolutionIsReadOnly = 1
    MeasurementResolution = 0.001
    CountDirectionIsReadOnly = 1
  MovementLimitsIsReadOnly = 1
  MovementLimits = InternalForPathControlledAxis
    VelocityIsReadOnly = 1
    Velocity:
      VelocityMax = 1000.0
    AccelerationIsReadOnly = 1
    Acceleration:
      AccelerationMax = 50000.0
      Acceleration = 50000.0
    DecelerationIsReadOnly = 1
    Deceleration:
      DecelerationMax = 50000.0
      Deceleration = 50000.0
    JerkIsReadOnly = 1
    Jerk = Advanced
      JerkAccelerationPositiveMin = 0.0
      JerkAccelerationPositiveMax = 1300000.0
      JerkAccelerationPositive = 1300000.0
      JerkAccelerationNegativeMin = 0.0
      JerkAccelerationNegativeMax = 1300000.0
      JerkAccelerationNegative = 1300000.0
      JerkDecelerationPositiveMin = 0.0
      JerkDecelerationPositiveMax = 1300000.0
      JerkDecelerationPositive = 1300000.0
      JerkDecelerationNegativeMin = 0.0
      JerkDecelerationNegativeMax = 1300000.0
      JerkDecelerationNegative = 1300000.0
    TorqueIsReadOnly = 1
    Torque = Basic
      TorqueMax = 1.67
      Torque = 1.67
Element gAxisQ4_SRr700_1 (Type=axis)  // Codian SR200-6/700Z20A [RobotID="CodianSR200p6r700Z20A" Version="6.8.0"]
  BaseTypeIsReadOnly = 1
  BaseType = Rotary
    MeasurementUnitIsReadOnly = 1
    MeasurementResolutionIsReadOnly = 1
    MeasurementResolution = 0.001
    CountDirectionIsReadOnly = 1
    CountDirection = Inverse
  MovementLimitsIsReadOnly = 1
  MovementLimits = InternalForPathControlledAxis
    VelocityIsReadOnly = 1
    Velocity:
      VelocityMax = 2000.0
      Velocity = 2000.0
    AccelerationIsReadOnly = 1
    Acceleration:
      AccelerationMax = 30000.0
      Acceleration = 30000.0
    DecelerationIsReadOnly = 1
    Deceleration:
      DecelerationMax = 30000.0
      Deceleration = 30000.0
    JerkIsReadOnly = 1
    Jerk = Advanced
      JerkAccelerationPositiveMin = 0.0
      JerkAccelerationPositiveMax = 1500000.0
      JerkAccelerationPositive = 1500000.0
      JerkAccelerationNegativeMin = 0.0
      JerkAccelerationNegativeMax = 1500000.0
      JerkAccelerationNegative = 1500000.0
      JerkDecelerationPositiveMin = 0.0
      JerkDecelerationPositiveMax = 1500000.0
      JerkDecelerationPositive = 1500000.0
      JerkDecelerationNegativeMin = 0.0
      JerkDecelerationNegativeMax = 1500000.0
      JerkDecelerationNegative = 1500000.0
    TorqueIsReadOnly = 1
    Torque = Basic
      TorqueMax = 1.11
      Torque = 1.11
```

### Config_4.mechanicalsystem - 5APC3100_KBU3_000/mappMotion/Codian_SRr700_1/Config_4.mechanicalsystem
```
Element MechSys_SRr700_1 (Type=mechanicalsystem)  // Codian SR200-6/700Z20A [RobotID="CodianSR200p6r700Z20A" Version="6.8.0"]
  TypeIsReadOnly = 1
  Type = Scara
    SubtypeIsReadOnly = 1
    Subtype:
      SceneViewerObject = ObjectID
        ID = 2750
      DescriptionIsReadOnly = 1
      Description:
        Dimensions:
          TranslationFromBaseToQ1IsReadOnly = 1
          TranslationFromBaseToQ1:
            Z = 177.0
          TranslationFromQ1ToQ2IsReadOnly = 1
          TranslationFromQ1ToQ2:
            XY = 425.0
            Z = 54.5
          TranslationFromQ2ToQZ:
            XY = 275.0
          TranslationFromQZToQCIsReadOnly = 1
          TranslationFromQZToQC:
            Z = -53.5
          TranslationFromQCToFlangeIsReadOnly = 1
          TranslationFromQCToFlange:
            Z = -30.0
        Offsets:
          JointAxisIsReadOnly = 1
          JointAxis[1]
          JointAxis[2]
          JointAxis[3]
          JointAxis[4]
        CountDirections:
          JointAxisIsReadOnly = 1
          JointAxis[1]
          JointAxis[2]
          JointAxis[3]
          JointAxis[4]
      TcpOrientation:
        Frames = Used
      WireFrameModel:
        Q1ToQ2:
          Distance = 5.0
        Q2ToQZ:
          Distance = 5.0
        QZToQC:
          Distance = 5.0
        QCToFlange:
          Distance = 5.0
        FlangeToTcp:
          Distance = 5.0
      DynamicModelIsReadOnly = 1
      InternalDynamicModelIsReadOnly = 1
      InternalDynamicModel = Used
        TypeIsReadOnly = 1
        Type = Codian SR200-6/700Z20A
        Row[1]:
          Value = 6
          Unit = 
          Description = Dynamic_model_variant
        Row[2]:
          Index = 1
          Value = 5.430278
          Unit = kg
          Description = m1
        Row[3]:
          Index = 2
          Value = 1.43276798974
          Unit = kgm
          Description = m1*rc1x
        Row[4]:
          Index = 3
          Value = 0.000467003908
          Unit = kgm
          Description = m1*rc1y
        Row[5]:
          Index = 4
          Value = 0.244802362518
          Unit = kgm
          Description = m1*rc1z
        Row[6]:
          Index = 5
          Value = 0.000123218047118
          Unit = kgm²
          Description = m1*rc1x*rc1y
        Row[7]:
          Index = 6
          Value = 0.0000210530031765
          Unit = kgm²
          Description = m1*rc1y*rc1z
        Row[8]:
          Index = 7
          Value = 0.0645906137456
          Unit = kgm²
          Description = m1*rc1x*rc1z
        Row[9]:
          Index = 8
          Value = 0.378032968558
          Unit = kgm²
          Description = m1*rc1x*rc1x
        Row[10]:
          Index = 9
          Value = 0.000000040162336088
          Unit = kgm²
          Description = m1*rc1y*rc1y
        Row[11]:
          Index = 10
          Value = 0.0110359353047
          Unit = kgm²
          Description = m1*rc1z*rc1z
        Row[12]:
          Index = 11
          Value = 0.022483
          Unit = kgm²
          Description = Jxx1
        Row[13]:
          Index = 12
          Value = 0.537046
          Unit = kgm²
          Description = Jyy1
        Row[14]:
          Index = 13
          Value = 0.523971
          Unit = kgm²
          Description = Jzz1
        Row[15]:
          Index = 14
          Value = 4.79047
          Unit = kg
          Description = m2
        Row[16]:
          Index = 15
          Value = 0.15806634812
          Unit = kgm
          Description = m2*rc2x
        Row[17]:
          Index = 16
          Value = -0.0115929374
          Unit = kgm
          Description = m2*rc2y
        Row[18]:
          Index = 17
          Value = 0.43553037052
          Unit = kgm
          Description = m2*rc2z
        Row[19]:
          Index = 18
          Value = -0.00038252056245
          Unit = kgm²
          Description = m2*rc2x*rc2y
        Row[20]:
          Index = 19
          Value = -0.00105398349666
          Unit = kgm²
          Description = m2*rc2y*rc2z
        Row[21]:
          Index = 20
          Value = 0.0143707601057
          Unit = kgm²
          Description = m2*rc2x*rc2z
        Row[22]:
          Index = 21
          Value = 0.00521555722257
          Unit = kgm²
          Description = m2*rc2x*rc2x
        Row[23]:
          Index = 22
          Value = 0.000028054908508
          Unit = kgm²
          Description = m2*rc2y*rc2y
        Row[24]:
          Index = 23
          Value = 0.0395966791662
          Unit = kgm²
          Description = m2*rc2z*rc2z
        Row[25]:
          Index = 24
          Value = 0.098841
          Unit = kgm²
          Description = Jxx2
        Row[26]:
          Index = 25
          Value = 0.309168
          Unit = kgm²
          Description = Jyy2
        Row[27]:
          Index = 26
          Value = 0.221562
          Unit = kgm²
          Description = Jzz2
        Row[28]:
          Index = 27
          Unit = kg
          Description = m3
        Row[29]:
          Index = 28
          Unit = kgm
          Description = m3*rc3x
        Row[30]:
          Index = 29
          Unit = kgm
          Description = m3*rc3y
        Row[31]:
          Index = 30
          Unit = kgm
          Description = m3*rc3z
        Row[32]:
          Index = 31
          Unit = kgm²
          Description = m3*rc3x*rc3y
        Row[33]:
          Index = 32
          Unit = kgm²
          Description = m3*rc3y*rc3z
        Row[34]:
          Index = 33
          Unit = kgm²
          Description = m3*rc3x*rc3z
        Row[35]:
          Index = 34
          Unit = kgm²
          Description = m3*rc3x*rc3x
        Row[36]:
          Index = 35
          Unit = kgm²
          Description = m3*rc3y*rc3y
        Row[37]:
          Index = 36
          Unit = kgm²
          Description = m3*rc3z*rc3z
        Row[38]:
          Index = 37
          Unit = kgm²
          Description = Jxx3
        Row[39]:
          Index = 38
          Unit = kgm²
          Description = Jyy3
        Row[40]:
          Index = 39
          Unit = kgm²
          Description = Jzz3
        Row[41]:
          Index = 40
          Value = 0.859593
          Unit = kg
          Description = m4
        Row[42]:
          Index = 41
          Unit = kgm
          Description = m4*rc4x
        Row[43]:
          Index = 42
          Unit = kgm
          Description = m4*rc4y
        Row[44]:
          Index = 43
          Value = 0.058800459165
          Unit = kgm
          Description = m4*rc4z
        Row[45]:
          Index = 44
          Unit = kgm²
          Description = m4*rc4x*rc4y
        Row[46]:
          Index = 45
          Unit = kgm²
          Description = m4*rc4y*rc4z
        Row[47]:
          Index = 46
          Unit = kgm²
          Description = m4*rc4x*rc4z
        Row[48]:
          Index = 47
          Unit = kgm²
          Description = m4*rc4x*rc4x
        Row[49]:
          Index = 48
          Unit = kgm²
          Description = m4*rc4y*rc4y
        Row[50]:
          Index = 49
          Value = 0.00402224540918
          Unit = kgm²
          Description = m4*rc4z*rc4z
        Row[51]:
          Index = 50
          Unit = kgm²
          Description = Jxx4
        Row[52]:
          Index = 51
          Unit = kgm²
          Description = Jyy4
        Row[53]:
          Index = 52
          Value = 0.000371
          Unit = kgm²
          Description = Jzz4
        Row[54]:
          Index = 53
          Value = 0.000135
          Unit = kgm²
          Description = JMotor1
        Row[55]:
          Index = 54
          Value = 0.000065
          Unit = kgm²
          Description = JMotor2
        Row[56]:
          Index = 55
          Value = 0.000055
          Unit = kgm²
          Description = JMotor3
        Row[57]:
          Index = 56
          Value = 0.00003
          Unit = kgm²
          Description = JMotor4
        Row[58]:
          Index = 57
          Value = 1.95
          Unit = Nms
          Description = dV1
        Row[59]:
          Index = 58
          Value = 0.477
          Unit = Nms
          Description = dV2
        Row[60]:
          Index = 59
          Value = 120.0
          Unit = Ns/m
          Description = dV3
        Row[61]:
          Index = 60
          Value = 0.0129
          Unit = Nms
          Description = dV4
        Row[62]:
          Index = 61
          Value = 13.6
          Unit = Nm
          Description = dC1
        Row[63]:
          Index = 62
          Value = 5.0
          Unit = Nm
          Description = dC2
        Row[64]:
          Index = 63
          Value = 35.0
          Unit = N
          Description = dC3
        Row[65]:
          Index = 64
          Value = 0.37
          Unit = Nm
          Description = dC4
      InternalDynamicLimits = Used
        TypeIsReadOnly = 1
        Type = Codian SR200-6/700Z20A
        GearboxLimits:
          Row[1]:
            Value = 6
            Unit = Variant
            Description = Variant of dynamic model
          Row[2]:
            Index = 1
            Value = 113.0
            Unit = Nm
            Description = Gearbox Drive 1 Output Torque Limit
          Row[3]:
            Index = 2
            Value = 44.0
            Unit = Nm
            Description = Gearbox Drive 2 Output Torque Limit
          Row[4]:
            Index = 3
            Value = 100.0
            Unit = Nm
            Description = Gearbox Drive 3 Output Torque Limit
          Row[5]:
            Index = 4
            Value = 1.3
            Unit = Nm
            Description = Gearbox Drive 4 Output Torque Limit
      ConditionalLimitReduction4Ax = Used
        ConditionalLimitReductionList4Ax[1] = ConditionReductionU
          LimitReductionInfluence4Ax:
            LimitRedInfluenceList[1] = Yes
            LimitRedInfluenceList[2]
            LimitRedInfluenceList[3]
            LimitRedInfluenceList[4]
          CondLimRedPoint[1]:
            SourceValue = 0.0
            LimitReductionInPercent = 0.0
          CondLimRedPoint[2]:
            SourceValue = 2.0
            LimitReductionInPercent = 0.0
          CondLimRedPoint[3]:
            SourceValue = 4.0
            LimitReductionInPercent = 0.0
          CondLimRedPoint[4]:
            SourceValue = 6.0
            LimitReductionInPercent = 58.3
          CondLimRedPoint[5]
          CondLimRedPoint[6]
          CondLimRedPoint[7]
          CondLimRedPoint[8]
          CondLimRedPoint[9]
          CondLimRedPoint[10]
        ConditionalLimitReductionList4Ax[2] = ConditionReductionU
          LimitReductionInfluence4Ax:
            LimitRedInfluenceList[1]
            LimitRedInfluenceList[2] = Yes
            LimitRedInfluenceList[3]
            LimitRedInfluenceList[4]
          CondLimRedPoint[1]:
            SourceValue = 0.0
            LimitReductionInPercent = 0.0
          CondLimRedPoint[2]:
            SourceValue = 2.0
            LimitReductionInPercent = 0.0
          CondLimRedPoint[3]:
            SourceValue = 4.0
            LimitReductionInPercent = 0.0
          CondLimRedPoint[4]:
            SourceValue = 6.0
            LimitReductionInPercent = 53.8
          CondLimRedPoint[5]
          CondLimRedPoint[6]
          CondLimRedPoint[7]
          CondLimRedPoint[8]
          CondLimRedPoint[9]
          CondLimRedPoint[10]
        ConditionalLimitReductionList4Ax[3] = ConditionReductionU
          LimitReductionInfluence4Ax:
            LimitRedInfluenceList[1]
            LimitRedInfluenceList[2]
            LimitRedInfluenceList[3] = Yes
            LimitRedInfluenceList[4]
          CondLimRedPoint[1]:
            SourceValue = 0.0
            LimitReductionInPercent = 0.0
          CondLimRedPoint[2]:
            SourceValue = 2.0
            LimitReductionInPercent = 0.0
          CondLimRedPoint[3]:
            SourceValue = 4.0
            LimitReductionInPercent = 0.0
          CondLimRedPoint[4]:
            SourceValue = 6.0
            LimitReductionInPercent = 69.2
          CondLimRedPoint[5]
          CondLimRedPoint[6]
          CondLimRedPoint[7]
          CondLimRedPoint[8]
          CondLimRedPoint[9]
          CondLimRedPoint[10]
        ConditionalLimitReductionList4Ax[4]
        ConditionalLimitReductionList4Ax[5]
      Couplings:
        LinearCoupling[1]:
          SourceAxisIsReadOnly = 1
          SourceAxis = 4
          SourceAxisUnitsIsReadOnly = 1
          SourceAxisUnits = 360.0
          TargetJointAxisIsReadOnly = 1
          TargetJointAxis = 3
          TargetJointAxisUnitsIsReadOnly = 1
          TargetJointAxisUnits = 20.0
      JointAxesPositionLimits:
        SingleJointAxisIsReadOnly[1] = 1
        SingleJointAxisIsReadOnly[2] = 1
        SingleJointAxisIsReadOnly[3] = 1
        SingleJointAxisIsReadOnly[4]
        JointAxis[1] = ConfigureJointAxesLimits
          LowerLimitMin = -132.0
          UpperLimitMax = 132.0
          LowerLimit = -132.0
          UpperLimit = 132.0
        JointAxis[2] = ConfigureJointAxesLimits
          LowerLimitMin = -150.0
          UpperLimitMax = 150.0
          LowerLimit = -150.0
          UpperLimit = 150.0
        JointAxis[3] = ConfigureJointAxesLimits
          LowerLimitMin = -190.0
          UpperLimitMax = 10.0
          LowerLimit = -190.0
          UpperLimit = 10.0
        JointAxis[4]
      MonitoringPoints = Standard
```

### Config_5.axesgroupfeature - 5APC3100_KBU3_000/mappMotion/Codian_SRr700_1/Config_5.axesgroupfeature
```
Element Feature_Programs_SRr700_1 (Type=axesgroupfeature)  // Codian SR200-6/700Z20A [RobotID="CodianSR200p6r700Z20A" Version="6.8.0"]
  Type:
    InitialSettings:
      AccuracyHoldDelays = User defined
        UserAxesDelay = 0.025
Element Feature_Jogging_SRr700_1 (Type=axesgroupfeature)  // Codian SR200-6/700Z20A [RobotID="CodianSR200p6r700Z20A" Version="6.8.0"]
  Type = Jogging
Element Feature_FeedForward_SRr700_1 (Type=axesgroupfeature)  // Codian SR200-6/700Z20A [RobotID="CodianSR200p6r700Z20A" Version="6.8.0"]
  Type = FeedForward
    RiseTime = 0.25
    Filter = AxisJerkTime
Element Feature_SharedBrakesSignals_SRr700_1 (Type=axesgroupfeature)  // Codian SR200-6/700Z20A [RobotID="CodianSR200p6r700Z20A" Version="6.8.0"]
  Type = SharedBrakesSignals
    BrakeComposite[1]:
      Axes:
        AxisRef[1] = gAxisQ3_SRr700_1
        AxisRef[2] = gAxisQ4_SRr700_1
      Output:
        AxisRef = gAxisQ4_SRr700_1
      Feedback:
        ActivationDelay = 0.08
        ReleaseDelay = 0.2
```

### Config_6.dynpartable - 5APC3100_KBU3_000/mappMotion/Codian_SRr700_1/Config_6.dynpartable
```
Element ProductLoad_1 (Type=dynpartable)
  Row[1]:
    Value = 2.5
    Unit = kg
    Description = Mass
  Row[2]:
    Index = 1
    Unit = m
    Description = Center of gravity - X direction
  Row[3]:
    Index = 2
    Unit = m
    Description = Center of gravity - Y direction
  Row[4]:
    Index = 3
    Unit = m
    Description = Center of gravity - Z direction
  Row[5]:
    Index = 4
    Unit = kg m^2
    Description = Moment of inertia about X
  Row[6]:
    Index = 5
    Unit = kg m^2
    Description = Moment of inertia about Y
  Row[7]:
    Index = 6
    Unit = kg m^2
    Description = Moment of inertia about Z
  Row[8]:
    Index = 1000
    Value = 1
    Unit = 
    Description = 0 (toolDynPar), 1 (productLoadPar)
```

### ComRobot.axesgroupfeature - 5APC3100_KBU3_000/mappMotion/ComRobot.axesgroupfeature
```
Element Feature_TrackingRobot (Type=axesgroupfeature)
  Type = Tracking
    MotionBehaviour:
      OutOfWorkspaceSynchronisation:
        Clearance = 10
      OutOfWorkspaceSychronized = AdjustedVelocity
        Clearance = 10
Element Feature_MFunctions (Type=axesgroupfeature)
  Type = MFunctions
    MFunction[1]:
      IndexType:
        Index = 16
      Blocking = Disabled
      InSimulation = Set
      PvMapping = ::APP_Robot1:M16
    MFunction[2]:
      IndexType:
        Index = 17
      Blocking = Disabled
      InSimulation = Set
      PvMapping = ::APP_Robot1:M17
    MFunction[3]:
      IndexType:
        Index = 32
      Blocking = Disabled
      InSimulation = Set
      PvMapping = ::APP_Robot1:M32
    MFunction[4]:
      IndexType:
        Index = 33
      Blocking = Disabled
      InSimulation = Set
      PvMapping = ::APP_Robot1:M33
    MFunction[5]:
      IndexType:
        Index = 34
      Blocking = Disabled
      InSimulation = Set
      PvMapping = ::APP_Robot1:M34
    MFunction[6]:
      IndexType:
        Index = 40
      Blocking = Disabled
      InSimulation = Set
      PvMapping = ::APP_Robot1:M40
Element Feature_PathDefRobot (Type=axesgroupfeature)
  Type = PathDefinitions
    PathDefinition[1]:
      Type:
        CalculatedIn = PCS
Element Feature_FrameHierachy (Type=axesgroupfeature)
  Type = FrameHierarchy
    FrameHierarchy = Custom
      FramePropertyMapping:
        BCS = RobotBase
      MCS:
        Frame[1]:
          Name = RobotBase
        Frame[2]:
          Name = UserFrame1
          Frame[1]:
            Name = FixedPlace
            Type:
              Translation:
                Y = 450
Element Feature_Selection (Type=axesgroupfeature)
  Type = TrackingFrameSelection
    Selectors:
      Selector[1]:
        Name = Infeed
        Filters:
          Filter[1]:
            TrackingPathRef[1] = gTrackingPathConveyor_1
          Filter[2] = SelectionArea
            Area[1]:
              Translation:
                X = -500
                Y = -500
                Z = -500
              Dimensions:
                Length = 800
                Width = 1000
                Height = 1000
          Filter[3] = AttributeMask
            Mask = 2#00000000000000000000000000000001
Element Feature_Programs (Type=axesgroupfeature)
  Type:
    DefaultLanguage = ST
```

### AxisAx_1.axis - 5APC3100_KBU3_000/mappMotion/Conveyor/AxisAx_1.axis
```
Element gAxis_Conveyor_1 (Type=axis)
  BaseType = LinearPeriodic
    PeriodSettings:
      Period = 100000.0
  MovementLimits = InternalForPathControlledAxis
    Position:
      LowerLimit = -8388608.0
      UpperLimit = 8388607.0
```

### Config_1.trackingpath - 5APC3100_KBU3_000/mappMotion/Conveyor/Config_1.trackingpath
```
Element gTrackingPathConveyor_2 (Type=trackingpath)  // Tracking Path with moving objects
  Type:
    MotionSource = Axis
      AxisRef = gAxis_Conveyor_2
    TrackingFrames:
      AutomaticCreation:
        Condition[1]:
          Distance = 160
          Position:
            Translation:
              Y = -125
        Condition[2]:
          Distance = 160
          Position:
            Translation:
              Y = 125
      AutomaticDeletion:
        Condition[1]:
          MinPosition = -100
          MaxPosition = 2200
  SceneViewerObject:
    VisualRepresentation = Conveyor belt
      Dimensions:
        Length = 2200
        Width = 450
        Height = 1
      Translation:
        Y = -150
        Z = -50
Element gTrackingPathConveyor_1 (Type=trackingpath)  // Tracking Path with moving objects
  Type:
    MotionSource = Axis
      AxisRef = gAxis_Conveyor_1
    TrackingFrames:
      AutomaticCreation:
        Condition[1]:
          Distance = 130
          Position:
            Translation:
              Y = -113
        Condition[2]:
          Distance = 130
          Position:
            Translation:
              Y = 113
      AutomaticDeletion:
        Condition[1]:
          MinPosition = -100
          MaxPosition = 2200
        Condition[2] = AfterDesynchronization
          AxesGroupRef = gAxesGroup_D4r1100R_1
  SceneViewerObject:
    VisualRepresentation = Conveyor belt
      Dimensions:
        Length = 2200
        Width = 450
        Height = 1
      Translation:
        Y = -150
        Z = -50
```

### Config_7.purevaxcfg - 5APC3100_KBU3_000/mappMotion/Conveyor/Config_7.purevaxcfg
```
Element PureVAxCfg_1 (Type=purevaxcfg)
  PureVAxis:
    AxisReference = gAxis_Conveyor_1
Element PureVAxCfg_2 (Type=purevaxcfg)
  PureVAxis:
    AxisReference = gAxis_Conveyor_2
    JerkFilter = JerkLimited
      JerkLimit = 1000.0
```

## Logical view

Binary libraries used (declarations not repeated): operator, runtime, astime, AsIecCon, standard, AsBrStr, sys_lib, AsArSdm, brsystem, FileIO, AsIODiag, DataObj, AsArProf, AsMem, AsIOAcc, AsEPL, ASMcDcs, AsBrMath, visapi, ArTextSys, AsSem, AsZip, AcpInvLib, MpCom 6.3.2, MpUserX 6.3.2, MpFile 6.3.2, MpRecipe 6.3.2, MpAlarmX 6.3.2, MpBase, CoTrace 6.3.1, MpServer 6.6.0, McBase 6.8.0, McAxGroup 6.8.0, McAcpAx 6.8.0, McAxis 6.8.0, McPathGen 6.8.0, McTrkPath 6.8.0, MpAxis 6.8.0, McProgInt 6.8.0, McPureVAx 6.8.0, McDS402Ax 6.8.0, MpRobotics 6.8.0, MpCnc 6.8.0, MpTool 6.8.0

### Global.typ
```iecst
TYPE
	ControlPanelInputs : 	STRUCT  (*Command Buttons*)
		Start : BOOL; (*Run a pick and place application demo*)
		Reset : BOOL; (*Stop Execute*)
		PickRate : REAL; (*Velocity for production [ppm]*)
	END_STRUCT;
	ControlPanelType : 	STRUCT  (*Control Panel*)
		Input : ControlPanelInputs; (*Buttons *)
	END_STRUCT;
END_TYPE
```

### Global.var
```iecst
VAR
	ControlPanel : ControlPanelType := (Input:=(PickRate:=60)); (*Machine interface (inputs/outputs)*)
END_VAR
```

### Conveyor.typ
```iecst
TYPE
	ConveyorStatesEnum :
		( (*State of the robot*)
		STATE_WAIT,
		STATE_RESET,
		STATE_POWER,
		STATE_HOME,
		STATE_PRODUCTION,
		STATE_ERROR
		);
END_TYPE
```

### Program Logical/Conveyor/APP_Conveyor1 (IEC) - Motion Belt

#### Variables.var - Local variables
```iecst
(*
MpAxisBasic function blocks used for Conveyor Handling*)
VAR
	Period : LREAL;
	LinkAxis : UDINT;
	LinkTrackingPath : UDINT;
	LastProductPosition : LREAL := 0;
	State : ConveyorStatesEnum;
	Reset : BOOL;
	Start : BOOL;
	SetVelocity : REAL;
	timeLast : UDINT;
	ProductGap : LREAL;
	Indexing : BOOL;
	Multipick : BOOL;
END_VAR
(*Ax Mngment Functions*)
VAR
	MC_Stop_0 : MC_Stop;
	MC_Reset_0 : MC_Reset;
	MC_Power_0 : MC_Power;
	MC_Home_0 : MC_Home;
	MC_MoveVelocity_0 : MC_MoveVelocity;
	MC_MoveAdditive_0 : MC_MoveAdditive;
	MC_ReadStatus_0 : MC_ReadStatus;
	MC_ReadActualPosition_0 : MC_ReadActualPosition;
END_VAR
(*
Tracking function*)
VAR
	MC_BR_TrackingFrameCreate_0 : MC_BR_TrackingFrameCreate;
	MC_BR_TrackingPathReset_0 : MC_BR_TrackingPathReset;
	MC_BR_TrackingPathReadStatus_0 : MC_BR_TrackingPathReadStatus;
	MC_BR_TrackingPathReadInfo_0 : MC_BR_TrackingPathReadInfo;
	MC_BR_TrackingFrameDelete_0 : MC_BR_TrackingFrameDelete;
	createCnt : USINT;
	RandomCreation : BOOL;
END_VAR
```

#### Init.st - Init code
```iecst
PROGRAM _INIT

	DefineLinks;

	// Set Default Parameters of the Tracking Frames
	MC_BR_TrackingFrameCreate_0.Parameters.Attribute	:= 0;
	MC_BR_TrackingFrameCreate_0.Parameters.Translation.X := 0.0;
	MC_BR_TrackingFrameCreate_0.Parameters.Translation.Y := 0.0;
	MC_BR_TrackingFrameCreate_0.Parameters.Translation.Z := 0.0;
	MC_BR_TrackingFrameCreate_0.Parameters.Orientation.Angle1 := 0.0;
	MC_BR_TrackingFrameCreate_0.Parameters.Orientation.Angle2 := 0.0;
	MC_BR_TrackingFrameCreate_0.Parameters.Orientation.Angle3 := 0.0;
	MC_BR_TrackingFrameCreate_0.Parameters.Orientation.Type := 0;

	MC_BR_TrackingFrameDelete_0.Mode :=  mcTRKFRM_DELETE_MOD_ALL;

	MC_Home_0.HomingMode := mcHOMING_DEFAULT;
	MC_ReadStatus_0.Enable := TRUE;
	MC_BR_TrackingPathReadInfo_0.Enable := TRUE;
	MC_BR_TrackingPathReadStatus_0.Enable := TRUE;
	MC_ReadActualPosition_0.Enable := TRUE;

END_PROGRAM
```

#### Cyclic.st - Cyclic code
```iecst
PROGRAM _CYCLIC
	DefineLinks;

	CASE State OF

		/////////////////////////////////////////////////////////////////////////////
		STATE_WAIT:
		/////////////////////////////////////////////////////////////////////////////
			IF  Start THEN
				State := STATE_RESET;
				MC_Power_0.Enable := FALSE;
			END_IF

		/////////////////////////////////////////////////////////////////////////////
		STATE_RESET:
		////////////////////////////////////////////////////////////////////////////
			MC_Reset_0.Execute := TRUE;
			MC_BR_TrackingPathReset_0.Execute := TRUE;

			IF MC_Reset_0.Done AND MC_BR_TrackingPathReset_0.Done THEN
				State := STATE_POWER;
			END_IF

		/////////////////////////////////////////////////////////////////////////////
		STATE_POWER:
		////////////////////////////////////////////////////////////////////////////
			MC_Power_0.Enable := TRUE;
			IF MC_Power_0.Status THEN
				State := STATE_HOME;
			END_IF

		/////////////////////////////////////////////////////////////////////////////
		STATE_HOME:
		////////////////////////////////////////////////////////////////////////////
			MC_Home_0.Execute := TRUE;
			IF MC_Home_0.Done THEN
				MC_MoveVelocity_0.Velocity := SetVelocity;
				MC_MoveVelocity_0.Acceleration := SetVelocity/10;
				MC_MoveVelocity_0.Deceleration := SetVelocity/10;

				MC_MoveAdditive_0.Distance := ProductGap;
				MC_MoveAdditive_0.Acceleration := SetVelocity*4;
				MC_MoveAdditive_0.Deceleration := SetVelocity*4;
				MC_MoveAdditive_0.Jerk := SetVelocity*2*10;
				MC_MoveAdditive_0.Velocity := 4*SetVelocity;

				IF NOT Indexing THEN
					MC_MoveVelocity_0.Execute := TRUE;
				ELSE
					MC_MoveAdditive_0.Execute := TRUE;
				END_IF
				timeLast := 0;
				State := STATE_PRODUCTION;
			END_IF

		///////////////////////////////////////////////////////////////////////////////
		STATE_PRODUCTION:
		///////////////////////////////////////////////////////////////////////////////

			IF NOT Indexing AND MC_MoveVelocity_0.Velocity <> SetVelocity AND MC_MoveVelocity_0.InVelocity THEN
				MC_MoveVelocity_0.Velocity := SetVelocity;
				MC_MoveVelocity_0.Execute := TRUE;
			END_IF

			timeLast := timeLast + 1;
			IF Indexing AND (UDINT_TO_REAL(timeLast * 2)/1000.0) >= (LREAL_TO_REAL(ProductGap) / SetVelocity) THEN
				timeLast := 0;
				MC_MoveAdditive_0.Execute := TRUE;
			END_IF

			IF MC_ReadStatus_0.Error OR MC_ReadStatus_0.ErrorStop THEN
				State := STATE_ERROR;

			ELSIF NOT Start THEN
				MC_Stop_0.Execute := TRUE;
				IF MC_Stop_0.Done THEN
					State := STATE_WAIT;
				END_IF
			END_IF

		///////////////////////////////////////////////////////////////////////////////
		STATE_ERROR:
		///////////////////////////////////////////////////////////////////////////////
			MC_Power_0.Enable := FALSE;
			MC_BR_TrackingPathReset_0.Execute := TRUE;

			IF ControlPanel.Input.Reset AND NOT MC_BR_TrackingPathReset_0.Busy THEN
				State := STATE_WAIT;
			END_IF
	END_CASE

	(* *************************************************************************************************************************** *)
	(* *************************************************************************************************************************** *)
	(* *************************************************************************************************************************** *)

	// Axis commands
	MC_MoveAdditive_0(Axis := LinkAxis);
	MC_MoveVelocity_0(Axis := LinkAxis);
	MC_Stop_0(Axis := LinkAxis);
	MC_Reset_0(Axis := LinkAxis);
	MC_Home_0(Axis := LinkAxis);
	MC_Power_0(Axis := LinkAxis);
	MC_ReadStatus_0(Axis := LinkAxis);
	MC_ReadActualPosition_0(Axis := LinkAxis);

	MC_MoveAdditive_0.Execute := FALSE;
	MC_MoveVelocity_0.Execute := FALSE;
	MC_Stop_0.Execute := FALSE;
	MC_Reset_0.Execute := FALSE;
	MC_Home_0.Execute := FALSE;
	MC_Power_0.Enable := MC_Power_0.Enable AND NOT MC_Power_0.Error;

	// Trackingpath commands
	MC_BR_TrackingFrameCreate_0(TrackingPath := LinkTrackingPath);
	MC_BR_TrackingFrameDelete_0(TrackingPath := LinkTrackingPath);
	MC_BR_TrackingPathReset_0(TrackingPath := LinkTrackingPath);
	MC_BR_TrackingPathReadStatus_0(TrackingPath := LinkTrackingPath);
	MC_BR_TrackingPathReadInfo_0(TrackingPath := LinkTrackingPath);

	MC_BR_TrackingFrameCreate_0.Execute := FALSE;
	MC_BR_TrackingFrameDelete_0.Execute := FALSE;
	MC_BR_TrackingPathReset_0.Execute := FALSE;

END_PROGRAM
```

#### DefineLinks.st
```iecst
ACTION DefineLinks:
	LinkTrackingPath := ADR(gTrackingPathConveyor_1);
	LinkAxis := ADR(gAxis_Conveyor_1);
	Period := 100000.0;

	Reset := ControlPanel.Input.Reset;
	Start := ControlPanel.Input.Start

	ProductGap := 130;
	SetVelocity := ProductGap / (ControlPanel.Input.PickRate / 60) / 2;

END_ACTION
```

#### DeviceActions.st - not listed in the package file held
```iecst
ACTION addNewObjects:

	// overflow handling
	IF MC_ReadActualPosition_0.Position < LastProductPosition THEN
		LastProductPosition := LastProductPosition - Period;
	END_IF

	IF MC_ReadActualPosition_0.Position <  LastProductPosition	+ ProductGap THEN
		RETURN;
	END_IF

	IF Multipick THEN
		MC_BR_TrackingFrameCreate_0.Parameters.Translation.Y := 80 - UDINT_TO_LREAL(createCnt MOD 2) * 160;
		createCnt := createCnt + 1;

		IF createCnt MOD 2 = 0 THEN
			LastProductPosition := MC_ReadActualPosition_0.Position;
		END_IF

	ELSE
		IF RandomCreation THEN
			MC_BR_TrackingFrameCreate_0.Parameters.Translation.Y := (UINT_TO_LREAL((TIM_musec()*10) MOD 160) - 80);
			MC_BR_TrackingFrameCreate_0.Parameters.Orientation.Angle3 := (UINT_TO_LREAL((TIM_musec()*10) MOD 178)-89);
		ELSE
			MC_BR_TrackingFrameCreate_0.Parameters.Translation.Y := 0;
			MC_BR_TrackingFrameCreate_0.Parameters.Orientation.Angle3 := 0;
		END_IF
		LastProductPosition := MC_ReadActualPosition_0.Position;
	END_IF

	// simulate two diffent product types
	MC_BR_TrackingFrameCreate_0.Parameters.Attribute := 2#0001;
	IF (TIM_ticks() MOD 2) = 1 THEN
		MC_BR_TrackingFrameCreate_0.Parameters.Attribute := 2#0011;
	END_IF;

	// Add frame in the buffer
	MC_BR_TrackingFrameCreate_0.Parameters.LatchedPath.Position := MC_ReadActualPosition_0.Position;
	MC_BR_TrackingFrameCreate_0.Execute	:= TRUE;

END_ACTION
```

### Program Logical/Conveyor/APP_Conveyor2 (IEC)

- Cyclic.st (reference to Logical/Conveyor/APP_Conveyor1/Cyclic.st)

- Init.st (reference to Logical/Conveyor/APP_Conveyor1/Init.st)

- Variables.var (reference to Logical/Conveyor/APP_Conveyor1/Variables.var)

#### DefineLinks.st
```iecst
ACTION DefineLinks:
	LinkTrackingPath := ADR(gTrackingPathConveyor_2);
	LinkAxis := ADR(gAxis_Conveyor_2);
	Period := 100000.0;

	Reset := ControlPanel.Input.Reset;
	Start := ControlPanel.Input.Start

	ProductGap := 160;
	SetVelocity := ProductGap / (ControlPanel.Input.PickRate / 60) / 2;

END_ACTION
```

### PickNPlace.st
```iecst
VAR CONSTANT
	UpperZLevel : LREAL := 10.0;	// Gripper up position
	LowerZLevel : LREAL := -10.0;	// Gripper down movement
END_VAR

VAR

	ParkPos				: McPointType := (Pos:=(X:=	  300, Y:= 100, Z:= 50));
	ParkPosRight		: McAxisTargetType :=(JointAxis:=[45, -90, -20, 0]);

	SynchPosUp			: McPointType := (Pos:=(X:=   0, Y:= 0, 			Z:= UpperZLevel));
	SynchPosDown		: McPointType := (Pos:=(X:=   0, Y:= 0, 			Z:= LowerZLevel));

	FrameIn : McTrkFrmIdentType;
END_VAR

PROGRAM _MAIN

	// Position init, reset frame in case of restart
	SetPCS(MachineFrame);
	MoveAR(ParkPosRight);
	SetProductLoad('ProductLoad_1');
	Feedrate(1000);
	MoveL(ParkPos);
	WaitEndMove();

	WaitUntil(TrackingFrameSelect(FrameIn,'Infeed'));				// hold interpreter until a new frame is available
	REPEAT

		TrackObjectR(FrameIn, SynchPosUp, 25, 25);					// track on product
		Relative();
		MoveLR(SynchPosDown);										// move to the take position
		WaitTime(0.075);											// Wait cause delay of gripper
		MoveLR(SynchPosUp);											// move up to change frame
		Absolute();

		TrackStopR(FixedPlace, SynchPosUp, 50, 50);					// Move to the fixed place Position
		Relative();
		MoveLR(SynchPosDown);										// move to the take position
		WaitTime(0.2);												// Wait cause delay of gripper
		MoveLR(SynchPosUp);											// move up to change frame
		Absolute();
		WaitALAP();

		IF NOT TrackingFrameSelect(FrameIn,'Infeed') THEN			// Need to stop, no objects left
			MoveLR(ParkPos);
			WaitEndMove();											// sync interpreter and program
			WaitUntil(TrackingFrameSelect(FrameIn,'Infeed'));		// hold interpreter until a new frame is available
		END_IF

	UNTIL FALSE END_REPEAT;

END_PROGRAM
```

### Program Logical/Robots/APP_Robot1

#### DefineLinks.st
```iecst
ACTION DefineLinks:

	// Define Link to the Robot & Conveyor
	NameAxesGroup	:= 'gAxesGroup_SRr500_1';
	LinkAxesGroup	:= ADR(gAxesGroup_SRr500_1);

	LinkTrackingPath := ADR(gTrackingPathConveyor_1);
	NameTrackingPath := 'gTrackingPathConveyor_1';
	LinkAxisTrackingPath := ADR(gAxis_Conveyor_1);

	Reset := ControlPanel.Input.Reset;
	Start :=
		(ControlPanel.Input.StartMultipick OR
		ControlPanel.Input.StartPickNPlace OR
		ControlPanel.Input.StartPlaceWithConditionalStop OR
		ControlPanel.Input.StartPrePalletizing OR
		ControlPanel.Input.StartSorting OR
		ControlPanel.Input.StartMultipickRandom);

	IF ControlPanel.Input.StartMultipickRandom THEN
		MC_BR_MoveProgram_X.Name := 'MultipickRandom.st';
	END_IF

	IF ControlPanel.Input.StartMultipick THEN
		MC_BR_MoveProgram_X.Name := 'Multipick.st';
	END_IF

	IF ControlPanel.Input.StartPickNPlace THEN
		MC_BR_MoveProgram_X.Name := 'PickNPlace.st';
	END_IF

	IF ControlPanel.Input.StartPlaceWithConditionalStop THEN
		MC_BR_MoveProgram_X.Name := 'PlaceWithConditionalStop.st';
	END_IF

	IF ControlPanel.Input.StartPrePalletizing THEN
		MC_BR_MoveProgram_X.Name := 'PrePalletizing.st';
	END_IF

	IF ControlPanel.Input.StartSorting THEN
		MC_BR_MoveProgram_X.Name := 'Sorting.st';
	END_IF

END_ACTION
```

Listed in the project but not available here: Logical/Conveyor/APP_Conveyor1/Exit.st, Logical/Conveyor/APP_Conveyor1/Exit.st
